FUNCTION_BLOCK ABSTRACT fb_MessageData IMPLEMENTS I_MessageData
VAR CONSTANT
{attribute 'hide'}
  STR_LEN       : UDINT := 524_288;
END_VAR
VAR
  _eCheck       : E_MESSAGE_CHECK;            // pointer check state

  _pFileRoot    : POINTER TO STRING(255);     // you decide (example in GVL_MSG.LOG_FILE)
  _pDirRoot     : POINTER TO STRING(255);     // see GVL_MSG.LOG_DIR

  _nMsgIndex    : REFERENCE TO UINT;          // Hypnos IS the only one in the village, if there are more you need more villages
  _nErrIndex    : REFERENCE TO UINT;          // Thanatos, Hypnos stern and more serious brother

  _dtLocalTime  : POINTER TO DT;
  _pMsgList     : POINTER TO ARRAY[1..GVL_MSG.MAX_MESSAGE] OF ST_Message; // attach your list here

	_rtrigReset   : Tc2_Standard.R_TRIG;
	_aWriteList   : ARRAY[1..GVL_MSG.MAX_MESSAGE] OF ST_Message;
	_sWriteData   : STRING(STR_LEN);
	_sNewLine     : STRING := '$N';
	_sTab         : STRING := '$T';
	_iCount, 
	_iStart, 
	_iEnd         : UINT;

	_fbCreateDir  : Tc2_System.FB_CreateDir;
	_sTmp         : STRING(256);
	_sFilename    : STRING(256);
	_sFolderDate  : STRING;
	_bFileCreated : BOOL;

	_fbFileOpen   : Tc2_System.FB_FileOpen;
	_fbFileWrite  : Tc2_System.FB_FileWrite;
	_fbFileClose  : Tc2_System.FB_FileClose;
END_VAR

METHOD Builder : BOOL // string concat for length > 255
VAR_INPUT
  pInString   : POINTER TO STRING;
  pOutString  : POINTER TO STRING(STR_LEN);
  Length      : UINT;
END_VAR
VAR
  Counter     : UDINT;
  pInWork     : POINTER TO BYTE;
  pOutWork    : POINTER TO BYTE;
END_VAR
pOutWork := pOutString;
pInWork := pInString;
Counter := 0;

(*check termination*)
WHILE (pOutWork^ <> 0) AND
      (Counter < STR_LEN+1)
DO
  Counter := Counter + 1;
  pOutWork := pOutWork + 1;
END_WHILE

(* append only if data fits into output *)
IF (Counter + Length < STR_LEN+1)
THEN

  (* append data *)
  FOR Counter := 1 TO Length
  DO
    pOutWork^ := pInWork^;
    pOutWork := pOutWork + 1;
    pInWork := pInWork + 1;
  END_FOR

  (* terminate *)
  pOutWork := pOutWork + 1;
  pOutWork^ := 0;
END_IF
END_METHOD

METHOD Check : BOOL
VAR_INPUT
END_VAR

IF NOT (_dtLocalTime <> 0)
THEN
  _eCheck       := E_MESSAGE_CHECK.MSG_CHECK_INVALID_POINTER_TIME;
  RETURN;
END_IF

IF NOT (_pMsgList <> 0)
THEN
  _eCheck       := E_MESSAGE_CHECK.MSG_CHECK_INVALID_POINTER_LIST;
  RETURN;
END_IF

IF NOT (_pFileRoot <> 0)
THEN
  _eCheck       := E_MESSAGE_CHECK.MSG_CHECK_INVALID_POINTER_ROOT_FILE;
  RETURN;
END_IF

IF NOT (_pDirRoot <> 0)
THEN
  _eCheck       := E_MESSAGE_CHECK.MSG_CHECK_INVALID_POINTER_ROOT_DIR;
  RETURN;
END_IF

IF NOT __ISVALIDREF(_nMsgIndex)
THEN
  _eCheck       := E_MESSAGE_CHECK.MSG_CHECK_INVALID_POINTER_MSG_IDX;
  RETURN;
END_IF

IF NOT __ISVALIDREF(_nErrIndex)
THEN
  _eCheck       := E_MESSAGE_CHECK.MSG_CHECK_INVALID_POINTER_ERR_IDX;
  RETURN;
END_IF


_eCheck         := E_MESSAGE_CHECK.MSG_CHECK_DONE;
Check           := TRUE;
END_METHOD

METHOD Device_to_String : string
VAR_INPUT
  eMsgDevice    : e_Device;
END_VAR
VAR
  sId                 : STRING := '_ID_';
  nId                 : UDINT;
END_VAR
IF (eMsgDevice < e_device.General)
THEN
  // below general case
  nId := TO_UDINT(eMsgDevice);
  sId := concat(sId, TO_STRING(nId));

  Device_to_String := concat(TO_STRING(eMsgDevice), sId);

ELSE
  IF (eMsgDevice >= e_Device.DataProduct)
  THEN
    nId := eMsgDevice MOD e_Device.DataProduct;
    sId := concat(sId, TO_STRING(nId));
 
    Device_to_String := concat(TO_STRING(e_Device.DataProduct), sId);

  ELSIF (eMsgDevice >= e_Device.Application)
  THEN
    nId := eMsgDevice MOD e_Device.Application;
    sId := concat(sId, TO_STRING(nId));
 
    Device_to_String := concat(TO_STRING(e_Device.Application), sId);

  ELSIF (eMsgDevice >= e_Device.Process)
  THEN
    nId := eMsgDevice MOD e_Device.Process;
    sId := concat(sId, TO_STRING(nId));
 
    Device_to_String := concat(TO_STRING(e_Device.Process), sId);

  ELSIF (eMsgDevice >= e_Device.Metrics)
  THEN
    nId := eMsgDevice MOD e_Device.Metrics;
    sId := concat(sId, TO_STRING(nId));
 
    Device_to_String := concat(TO_STRING(e_device.Metrics), sId);

  ELSIF (eMsgDevice >= e_device.XfcAxis)
  THEN
    nId := eMsgDevice MOD e_device.XfcAxis;
    sId := concat(sId, TO_STRING(nId));
 
    Device_to_String := concat(TO_STRING(e_device.XfcAxis), sId);

  ELSIF (eMsgDevice >= e_device.Axis)
  THEN
    nId := eMsgDevice MOD e_device.Axis;
    sId := concat(sId, TO_STRING(nId));
 
    Device_to_String := concat(TO_STRING(e_device.Axis), sId);

  ELSIF (eMsgDevice >= e_device.NciChannelCtrl)
  THEN
    nId := eMsgDevice MOD e_device.NciChannelCtrl;
    sId := concat(sId, TO_STRING(nId));
 
    Device_to_String := concat(TO_STRING(e_device.NciChannelCtrl), sId);

  ELSIF (eMsgDevice >= e_device.NciChannel)
  THEN
    nId := eMsgDevice MOD e_device.NciChannel;
    sId := concat(sId, TO_STRING(nId));
 
    Device_to_String := concat(TO_STRING(e_device.NciChannel), sId);

  ELSIF (eMsgDevice >= e_Device.Camming)
  THEN
    nId := eMsgDevice MOD e_Device.Camming;
    sId := concat(sId, TO_STRING(nId));
 
    Device_to_String := concat(TO_STRING(e_device.Camming), sId);

  ELSIF (eMsgDevice >= e_Device.XtsStation)
  THEN
    nId := eMsgDevice MOD e_Device.XtsStation;
    sId := concat(sId, TO_STRING(nId));
 
    Device_to_String := concat(TO_STRING(e_device.XtsStation), sId);

  ELSIF (eMsgDevice >= e_Device.XfcTouchProbe)
  THEN
    nId := eMsgDevice MOD e_Device.XfcTouchProbe;
    sId := concat(sId, TO_STRING(nId));
 
    Device_to_String := concat(TO_STRING(e_device.XfcTouchProbe), sId);

  ELSIF (eMsgDevice >= e_Device.XfcTriggerBox)
  THEN
    nId := eMsgDevice MOD e_Device.XfcTriggerBox;
    sId := concat(sId, TO_STRING(nId));
 
    Device_to_String := concat(TO_STRING(e_device.XfcTriggerBox), sId);

  ELSIF (eMsgDevice >= e_Device.XtsTransportUnit)
  THEN
    nId := eMsgDevice MOD e_Device.XtsTransportUnit;
    sId := concat(sId, TO_STRING(nId));
 
    Device_to_String := concat(TO_STRING(e_device.XtsTransportUnit), sId);

  ELSIF (eMsgDevice >= e_Device.MoverCtrl)
  THEN
    nId := eMsgDevice MOD e_Device.MoverCtrl;
    sId := concat(sId, TO_STRING(nId));
 
    Device_to_String := concat(TO_STRING(e_device.MoverCtrl), sId);

  ELSIF (eMsgDevice >= e_Device.Mover)
  THEN
    nId := eMsgDevice MOD e_Device.Mover;
    sId := concat(sId, TO_STRING(nId));
 
    Device_to_String := concat(TO_STRING(e_device.Mover), sId);

  ELSIF (eMsgDevice >= e_Device.XpuCtrl)
  THEN
    nId := eMsgDevice MOD e_Device.XpuCtrl;
    sId := concat(sId, TO_STRING(nId));
 
    Device_to_String := concat(TO_STRING(e_device.XpuCtrl), sId);

  ELSIF (eMsgDevice >= e_Device.Xpu)
  THEN
    nId := eMsgDevice MOD e_Device.Xpu;
    sId := concat(sId, TO_STRING(nId));
 
    Device_to_String := concat(TO_STRING(e_device.Xpu), sId);

  ELSIF (eMsgDevice >= e_Device.CaGroup)
  THEN
    nId := eMsgDevice MOD e_Device.CaGroup;
    sId := concat(sId, TO_STRING(nId));
 
    Device_to_String := concat(TO_STRING(e_device.CaGroup), sId);

  ELSIF (eMsgDevice >= e_Device.General)
  THEN
    nId := eMsgDevice MOD e_Device.General;
    sId := concat(sId, TO_STRING(nId));
 
    Device_to_String := concat(TO_STRING(e_device.General), sId);

  ELSE
    Device_to_String := TO_STRING(eMsgDevice);
  END_IF
END_IF
END_METHOD

PROPERTY DirRoot : POINTER to string(255)
SET
_pDirRoot := DirRoot;
END_SET
END_PROPERTY

PROPERTY ErrorIndex : reference to uint
SET
_nErrIndex  REF= ErrorIndex;
END_SET
END_PROPERTY

PROPERTY FileRoot : pointer to string(255)
SET
_pFileRoot := FileRoot;
END_SET
END_PROPERTY

METHOD FolderDate : STRING
VAR_INPUT
	LocalTime   : POINTER TO DT;
END_VAR
VAR
	sTmp        : STRING;
END_VAR
IF NOT (LocalTime <> 0)
THEN
	FolderDate := 'NULL';
	RETURN;
END_IF

sTmp := DT_TO_STRING(LocalTime^);

// cut off #dt literal
sTmp := right(sTmp, len(sTmp)-3);

sTmp := replace(sTmp, '_', 1, 5);
sTmp := replace(sTmp, '_', 1, 8);

sTmp := left(sTmp,10);	// year_month_day

FolderDate := sTmp;
END_METHOD

PROPERTY LocalTime : pointer to DT
SET
_dtLocalTime := LocalTime;
END_SET
END_PROPERTY

PROPERTY MessageIndex : reference to uint
SET
_nMsgIndex   REF= MessageIndex;
END_SET
END_PROPERTY

PROPERTY MsgList : pointer to ARRAY[1..GVL_MSG.MAX_MESSAGE] OF st_message
SET
_pMsgList := MsgList;
END_SET
END_PROPERTY

METHOD StringLen : UINT // 	string length for len > 255
VAR_INPUT
  pInString		: POINTER TO STRING(STR_LEN);
END_VAR
VAR
	Counter			: UINT;
	pInWork			: POINTER TO BYTE;
END_VAR
pInWork := pInString;
Counter := 0;

WHILE (pInWork^ <> 0) AND
			(Counter < STR_LEN)
DO
	Counter := Counter + 1;
	pInWork := pInWork + 1;
END_WHILE

StringLen := Counter;
END_METHOD

METHOD WriteData  : e_progress
VAR_INPUT
  bExecute        : BOOL;
END_VAR
VAR_INST
  _eState         : e_progress;
  _bError         : BOOL;
  _nErrorId       : UDINT;
END_VAR
IF NOT bExecute
THEN
  _eState                     := E_PROGRESS.PROGRESS_INIT;
END_IF

CASE _eState 
OF

	E_PROGRESS.PROGRESS_INIT:
		_fbFileOpen.bExecute      := FALSE;
		_fbFileWrite.bExecute	    := FALSE;
		_fbFileClose.bExecute	    := FALSE;

		IF bExecute
		THEN
      _nErrorId               := 0;
      _eState                 := E_PROGRESS.PROGRESS_BUSY;
		END_IF

	E_PROGRESS.PROGRESS_BUSY:
		_fbFileOpen.bExecute      := TRUE;

    IF _fbFileOpen.bError
    THEN
		  _fbFileOpen.bExecute    := FALSE;
      _nErrorId               := _fbFileOpen.nErrId;
      _eState                 := E_PROGRESS.PROGRESS_ERROR;

		ELSIF _fbFileOpen.bBusy
		THEN
      _eState                 := E_PROGRESS.PROGRESS_PREPARE;
		END_IF

	E_PROGRESS.PROGRESS_PREPARE:
		IF NOT _fbFileOpen.bBusy
		THEN
		  _fbFileOpen.bExecute    := FALSE;
			_fbFileWrite.bExecute   := TRUE;
      _eState                 := E_PROGRESS.PROGRESS_STARTUP;
		END_IF

	E_PROGRESS.PROGRESS_STARTUP:
    IF _fbFileWrite.bError
    THEN
			_fbFileWrite.bExecute   := FALSE;
      _nErrorId               := _fbFileWrite.nErrId;
      _eState                 := E_PROGRESS.PROGRESS_ERROR;

		ELSIF _fbFileWrite.bBusy
		THEN
      _eState                 := E_PROGRESS.PROGRESS_CHECK;
		END_IF

	E_PROGRESS.PROGRESS_CHECK:
		IF NOT _fbFileWrite.bBusy
		THEN
			_fbFileWrite.bExecute   := FALSE;
			_fbFileClose.bExecute   := TRUE;
      _eState                 := E_PROGRESS.PROGRESS_OCCUPIED;
		END_IF

	E_PROGRESS.PROGRESS_OCCUPIED:
    IF _fbFileClose.bError
    THEN
			_fbFileClose.bExecute   := FALSE;
      _nErrorId               := _fbFileClose.nErrId;
      _eState                 := E_PROGRESS.PROGRESS_ERROR;

		ELSIF _fbFileClose.bBusy
		THEN
      _eState                 := E_PROGRESS.PROGRESS_WORKING;
		END_IF

	E_PROGRESS.PROGRESS_WORKING:
		IF NOT _fbFileClose.bBusy
		THEN
			_fbFileClose.bExecute   := FALSE;
      _eState                 := E_PROGRESS.PROGRESS_DONE;
		END_IF
END_CASE


_fbFileOpen(
	sNetId:= , 
	sPathName:= _sFilename, 
	nMode:= FOPEN_MODEAPPEND OR FOPEN_MODEPLUS, 
	ePath:= PATH_GENERIC, 
	bExecute:= , 
	tTimeout:= T#10S, 
	bBusy=> , 
	bError=> , 
	nErrId=> , 
	hFile=> );

_fbFileWrite(
	sNetId:= , 
	hFile:= _fbFileOpen.hFile, 
	pWriteBuff:= ADR(_sWriteData), 
	cbWriteLen:= StringLen(ADR(_sWriteData)), 
	bExecute:= , 
	tTimeout:= T#10S, 
	bBusy=> , 
	bError=> , 
	nErrId=> , 
	cbWrite=> );

_fbFileClose(
	sNetId:= , 
	hFile:= _fbFileOpen.hFile, 
	bExecute:= , 
	tTimeout:= T#10S, 
	bBusy=> , 
	bError=> , 
	nErrId=> );

WriteData                     := _eState;
END_METHOD

END_FUNCTION_BLOCK

(* stored: Version 1.1.0.1
   POU fb_MessageData: Id {a6523f69-11be-4d44-a4e8-a8cdf6e59115}, SpecialFunc None
   Folder methods: Id {3dd7c8c4-0295-4e95-a801-983a245d2b7e}
   Folder properties: Id {37931ec5-8974-4db8-800c-832a5c8dd085}
   Method Builder: Id {c9561732-75b0-49ca-994a-77c64da760e6}
   Method Check: Id {b8a94b81-a325-4a55-8c76-d21d1bf6e45b}
   Method Device_to_String: Id {c4df82e6-06e9-458b-8675-2ae811f81a78}
   Property DirRoot: Id {7632cf51-d8a5-4b34-b0dd-cf27f49f3e81}
   Set Set: Id {fea85b73-0f61-4326-ba4f-c96f3398fe29}
   Property ErrorIndex: Id {40d116ce-c024-464c-994d-39c70dbde236}
   Set Set: Id {e6cd432b-5f9c-4534-8357-c62c61057155}
   Property FileRoot: Id {77e52297-39ee-49ff-bbe9-9575de067738}
   Set Set: Id {fd34aecd-eb33-46c3-9b7d-ca1cb02eaad2}
   Method FolderDate: Id {a57b1eb3-be3b-418f-be44-0bdeaa328468}
   Property LocalTime: Id {a15eeb2b-2fd1-42bd-bab0-31c596e0dedb}
   Set Set: Id {a8fc14cd-3d55-4d02-8a2f-6c167a473054}
   Property MessageIndex: Id {60143795-d3a6-455b-881b-f188e6bce075}
   Set Set: Id {effb092d-e9be-4d6d-a6ec-78a7b82c798a}
   Property MsgList: Id {9c2582e0-35d0-4ec2-9afd-d94acefaf83e}
   Set Set: Id {4380812f-9549-4ee0-bf26-34dc2482e273}
   Method StringLen: Id {a5368eff-7928-4bec-a3fc-38002f2aaf13}
   Method WriteData: Id {52743494-f79a-46c2-8d37-9a73f23c5b7b} *)
